INTERFACE ITF_LinkedList_Master EXTENDS ITF_LinkedList_Node

METHOD mListAdd : BOOL
VAR_INPUT
	itfNode:	ITF_LinkedList_Node;
END_VAR
END_METHOD

METHOD mListRemove : BOOL
VAR_INPUT
	itfNode:	ITF_LinkedList_Node;
END_VAR
END_METHOD

END_INTERFACE

(* stored: Version 1.1.0.1, ProductVersion 3.1.4024.12
   Itf ITF_LinkedList_Master: Id {af4fff4a-9016-4b05-8cb2-d5290d14c357}
   Method mListAdd: Id {a7d15d52-bf24-4b5f-b776-2ea30de0bc0c}
   Method mListRemove: Id {d51da422-89c6-4f99-aa46-9200061d4fd7} *)
